// This function has been automatically generated from the project information.
{attribute 'signature_flag' := '1073741824'}
{attribute 'TcGenerated'}
{attribute 'no-analysis'}
FUNCTION F_GetVersion : ST_LibVersion
VAR_INPUT
	
END_VAR

F_GetVersion.iMajor := 1;
F_GetVersion.iMinor := 1;
F_GetVersion.iBuild := 4;
F_GetVersion.iRevision := 0;
F_GetVersion.sVersion := '1.1.4';
F_GetVersion.nFlags := 0;

END_FUNCTION

(* stored: Version 1.1.0.1
   POU F_GetVersion: Id {0546d28b-c038-4d52-987a-248effc4f0cc}, SpecialFunc None *)
